// TIA Portal V18 export
FUNCTION_BLOCK "AccessControl"   // FB7, LAD
{ S7_Optimized_Access := 'TRUE' }
VERSION : 0.1
// stored: AutoNumber true, IsIECCheckEnabled false, IsRetainMemResEnabled false, MemoryReserve 100, SetENOAutomatically false, UDAEnableTagReadback false
   VAR_INPUT
      SearchStatus : Int;   // 0:未搜索;1:搜索中;2:搜索完成;
      RunArea : Bool;
      ACC_Ready : Bool;
      ACC_Run : Bool;
      ACC_StopBeam : Bool;
      Key : Bool;
      keyControl : Bool;
      Interlock : Bool;
      DoseAttenuation_Time : Time := T#1m;
      StartAlarm_Time : Time := T#2m;
   END_VAR
   VAR_OUTPUT
      StartAlarm : Bool;
      NoEntry : Bool;
      RestrictedEntry : Bool;
      ControlEntry : Bool;
   END_VAR
   VAR_IN_OUT
      AreaReady : Bool;
      BeamAllowed : Bool;
   END_VAR
   VAR
      State : Int;   // 0:禁止进入;1:限制进入;2:控制进入
      DoseAttenuation_Timer { S7_SetPoint := 'True'} : TON_TIME;
      StartAlarm_Timer { S7_SetPoint := 'True'} : TON_TIME;
   END_VAR
   VAR_TEMP   // added for the SCL form of the ladder/FBD networks
      _w1 : Bool;
   END_VAR
BEGIN

REGION Network 1
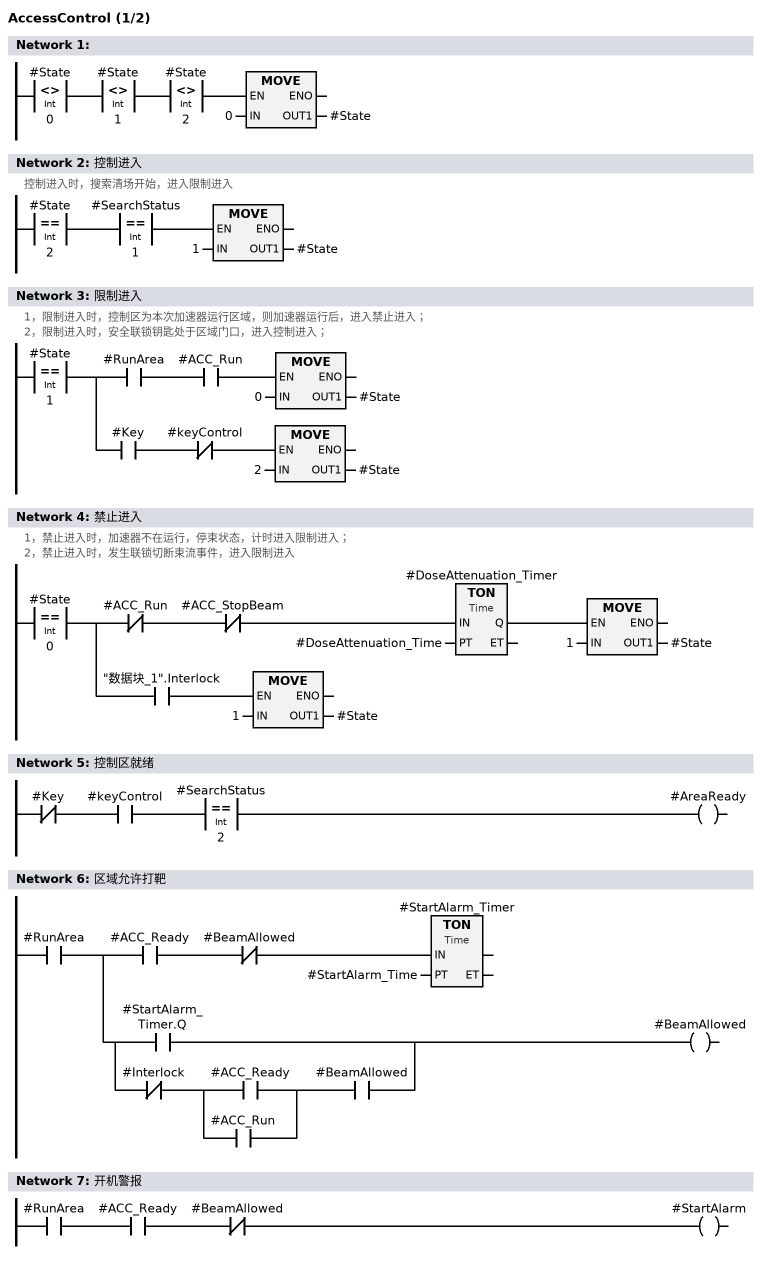
   RUNG wire#powerrail
      { S7_Templates := "SrcType := Int" } NE_Contact(in1 := #State, in2 := 0)
      { S7_Templates := "SrcType := Int" } NE_Contact(in1 := #State, in2 := 1)
      { S7_Templates := "SrcType := Int" } NE_Contact(in1 := #State, in2 := 2)
      Move(in := 0, out1 => #State)
   END_RUNG
   // the same network as SCL:
   IF (#State <> 0) AND (#State <> 1) AND (#State <> 2) THEN #State := 0; END_IF;
END_REGION

REGION Network 2: 控制进入
   // 控制进入时，搜索清场开始，进入限制进入
   RUNG wire#powerrail
      { S7_Templates := "SrcType := Int" } EQ_Contact(in1 := #State, in2 := 2)
      { S7_Templates := "SrcType := Int" } EQ_Contact(in1 := #SearchStatus, in2 := 1)
      Move(in := 1, out1 => #State)
   END_RUNG
   // the same network as SCL:
   IF (#State = 2) AND (#SearchStatus = 1) THEN #State := 1; END_IF;
END_REGION

REGION Network 3: 限制进入
   // 1，限制进入时，控制区为本次加速器运行区域，则加速器运行后，进入禁止进入；
   // 2，限制进入时，安全联锁钥匙处于区域门口，进入控制进入；
   RUNG wire#powerrail
      { S7_Templates := "SrcType := Int" } EQ_Contact(in1 := #State, in2 := 1)
      wire#w1
      Contact( #RunArea )
      Contact( #ACC_Run )
      Move(in := 0, out1 => #State)
   END_RUNG
   RUNG wire#w1
      Contact( #Key )
      I_Contact( #keyControl )
      Move(in := 2, out1 => #State)
   END_RUNG
   // the same network as SCL:
   #_w1 := #State = 1;
   IF #_w1 AND #RunArea AND #ACC_Run THEN #State := 0; END_IF;
   IF #_w1 AND #Key AND NOT #keyControl THEN #State := 2; END_IF;
END_REGION

REGION Network 4: 禁止进入
   // 1，禁止进入时，加速器不在运行，停束状态，计时进入限制进入；
   // 2，禁止进入时，发生联锁切断束流事件，进入限制进入
   RUNG wire#powerrail
      { S7_Templates := "SrcType := Int" } EQ_Contact(in1 := #State, in2 := 0)
      wire#w1
      I_Contact( #ACC_Run )
      I_Contact( #ACC_StopBeam )
      { S7_Templates := "time_type := Time" } #DoseAttenuation_Timer.TON(pt := #DoseAttenuation_Time, et =>)
      Move(in := 1, out1 => #State)
   END_RUNG
   RUNG wire#w1
      Contact( "数据块_1".Interlock )
      Move(in := 1, out1 => #State)
   END_RUNG
   // the same network as SCL:
   #_w1 := #State = 0;
   #DoseAttenuation_Timer(IN := #_w1 AND NOT #ACC_Run AND NOT #ACC_StopBeam, PT := #DoseAttenuation_Time);   // TON
   IF #DoseAttenuation_Timer.Q THEN #State := 1; END_IF;
   IF #_w1 AND "数据块_1".Interlock THEN #State := 1; END_IF;
END_REGION

REGION Network 5: 控制区就绪
   RUNG wire#powerrail
      I_Contact( #Key )
      Contact( #keyControl )
      { S7_Templates := "SrcType := Int" } EQ_Contact(in1 := #SearchStatus, in2 := 2)
      Coil( #AreaReady )
   END_RUNG
   // the same network as SCL:
   #AreaReady := NOT #Key AND #keyControl AND (#SearchStatus = 2);
END_REGION

REGION Network 6: 区域允许打靶
   RUNG wire#powerrail
      Contact( #RunArea )
      wire#w1
      Contact( #ACC_Ready )
      I_Contact( #BeamAllowed )
      { S7_Templates := "time_type := Time" } #StartAlarm_Timer.TON(pt := #StartAlarm_Time, et =>)
   END_RUNG
   RUNG wire#w1
      Contact( #StartAlarm_Timer.Q )
      wire#w2
      Coil( #BeamAllowed )
   END_RUNG
   RUNG wire#w1
      I_Contact( #Interlock )
      wire#w3
      Contact( #ACC_Ready )
      wire#w4
      Contact( #BeamAllowed )
   END_RUNG wire#w2
   RUNG wire#w3
      Contact( #ACC_Run )
   END_RUNG wire#w4
   // the same network as SCL:
   #StartAlarm_Timer(IN := #RunArea AND #ACC_Ready AND NOT #BeamAllowed, PT := #StartAlarm_Time);   // TON
   #BeamAllowed := #RunArea AND (#StartAlarm_Timer.Q OR (NOT #Interlock AND (#ACC_Ready OR #ACC_Run) AND #BeamAllowed));
END_REGION

REGION Network 7: 开机警报
   RUNG wire#powerrail
      Contact( #RunArea )
      Contact( #ACC_Ready )
      I_Contact( #BeamAllowed )
      Coil( #StartAlarm )
   END_RUNG
   // the same network as SCL:
   #StartAlarm := #RunArea AND #ACC_Ready AND NOT #BeamAllowed;
END_REGION

REGION Network 8
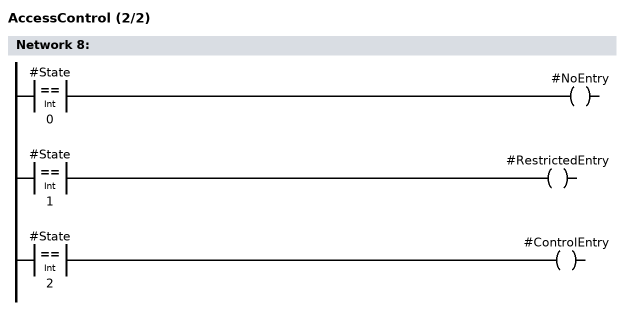
   RUNG wire#powerrail
      { S7_Templates := "SrcType := Int" } EQ_Contact(in1 := #State, in2 := 0)
      Coil( #NoEntry )
   END_RUNG
   RUNG wire#powerrail
      { S7_Templates := "SrcType := Int" } EQ_Contact(in1 := #State, in2 := 1)
      Coil( #RestrictedEntry )
   END_RUNG
   RUNG wire#powerrail
      { S7_Templates := "SrcType := Int" } EQ_Contact(in1 := #State, in2 := 2)
      Coil( #ControlEntry )
   END_RUNG
   // the same network as SCL:
   #NoEntry := #State = 0;
   #RestrictedEntry := #State = 1;
   #ControlEntry := #State = 2;
END_REGION
END_FUNCTION_BLOCK
